// TIA Portal V17 export
// export: Created 2025-01-08T13:55:37.6117632Z, ExportSetting WithDefaults, DisplayName Totally Integrated Automation Portal, DisplayVersion V17, DisplayName TIA Portal Openness, DisplayVersion V17, DisplayName TIA Portal Version Control Interface, DisplayVersion V17, DisplayName SINAMICS Startdrive Advanced, DisplayVersion V17 Update2, DisplayName SINAMICS Startdrive G130, G150, S120, S150, SINAMICS MV, S210, DisplayVersion V17 Update2, DisplayName SINAMICS Startdrive G110M, G120, G120C, G120D, G120P, G115D, DisplayVersion V17 Update2, DisplayName STEP 7 Professional, DisplayVersion V17, DisplayName STEP 7 Safety, DisplayVersion V17, DisplayName WinCC Advanced, DisplayVersion V17
TYPE "HSMMachineParaMask7"
// stored: IsFailsafeCompliant false
   STRUCT
      MPARA_I_Reserve_26 : Bool;
      MPARA_I_Reserve_27 : Bool;
      MPARA_I_Reserve_28 : Bool;
      MPARA_I_Reserve_29 : Bool;
      MPARA_I_Reserve_30 : Bool;
      MPARA_I_Reserve_31 : Bool;
      MPARA_I_Reserve_32 : Bool;
      MPARA_I_Reserve_33 : Bool;
      MPARA_I_Reserve_34 : Bool;
      MPARA_I_Reserve_35 : Bool;
      MPARA_I_Reserve_36 : Bool;
      MPARA_I_Reserve_37 : Bool;
      MPARA_I_Reserve_38 : Bool;
      MPARA_I_Reserve_39 : Bool;
      MPARA_I_Reserve_40 : Bool;
      MPARA_I_Reserve_41 : Bool;
   END_STRUCT;
END_TYPE
